// TIA Portal V17 export
// export: Created 2024-09-02T12:49:56.4347094Z, ExportSetting WithDefaults, DisplayName Totally Integrated Automation Portal, DisplayVersion V17, DisplayName TIA Portal Openness, DisplayVersion V17, DisplayName TIA Portal Version Control Interface, DisplayVersion V17, DisplayName STEP 7 Professional, DisplayVersion V17, DisplayName STEP 7 Safety, DisplayVersion V17, DisplayName WinCC Professional, DisplayVersion V17
FUNCTION "SysFC_Type_Change" : Void   // FC260, LAD
TITLE = Type change / Typwechsel
{ S7_Optimized_Access := 'TRUE' }
AUTHOR : OlegFuehrus
FAMILY : Typwechsel
NAME : Typwechsel
VERSION : 0.1
// stored: AutoNumber true, IsIECCheckEnabled false, SetENOAutomatically false, UDAEnableTagReadback false
   VAR_INPUT
      i_Start : Bool;   // Start Auswertung / Start evaluation
      i_Quit : Bool;   // Tywechsel Quitt / Tywechsel Quitt
      i_Reset : Bool;   // Speicher loeschen / Clear memory
      i_Data : Variant;   // Daten (max 64 Byte) / Data (max 64 Byte)
   END_VAR
   VAR_OUTPUT
      "o_Type Change" : Bool;   // Typwechsel / Type change
      "o_no Type Change" : Bool;   // kein Typwechsel / no type change
      "o_Data Fault" : Bool;   // Fehler Parameter / Error Parameter
   END_VAR
   VAR_IN_OUT
      io_IF_TypeChange : "TypeTypeChange";   // Interface Typwechsel / Interface type change
   END_VAR
   VAR_TEMP
      t_VKE0 : Bool;
      t_VKE1 : Bool;
      t_RetVal : Int;
      t_TempDInt : DInt;
      t_DataFault : Bool;
   END_VAR
   VAR_TEMP   // added for the SCL form of the ladder/FBD networks
      _w1 : Bool;
   END_VAR
BEGIN

REGION Network 1: INIT
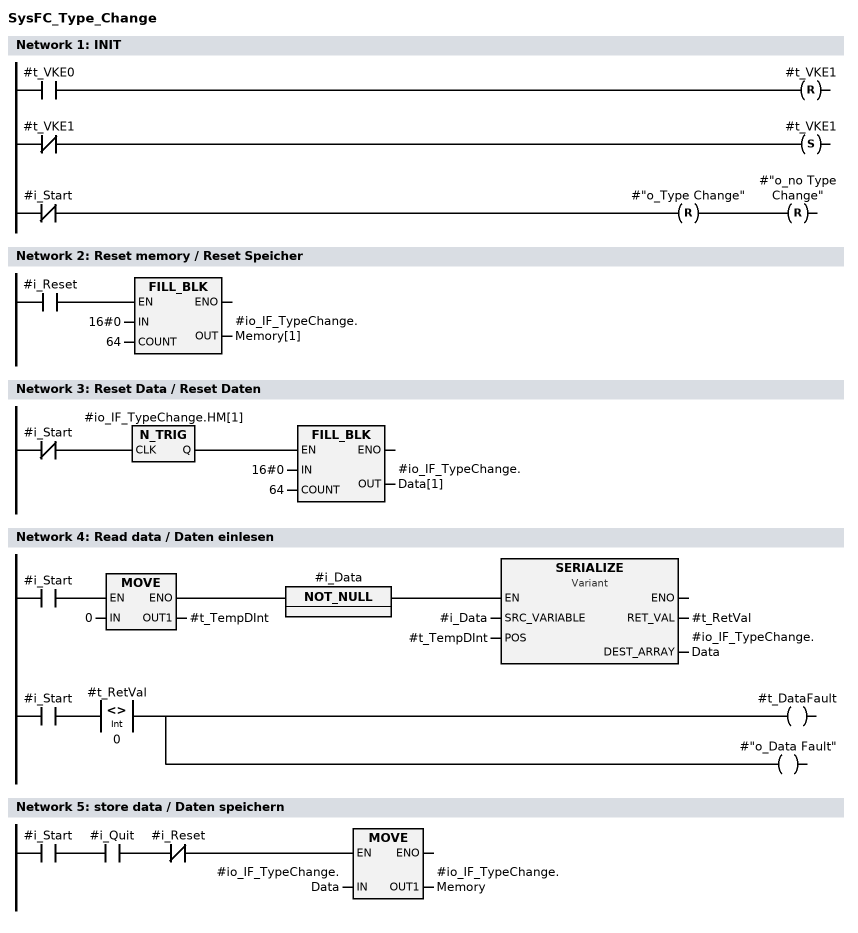
   RUNG wire#powerrail
      Contact( #t_VKE0 )
      R_Coil( #t_VKE1 )
   END_RUNG
   RUNG wire#powerrail
      I_Contact( #t_VKE1 )
      S_Coil( #t_VKE1 )
   END_RUNG
   RUNG wire#powerrail
      I_Contact( #i_Start )
      R_Coil( #"o_Type Change" )
      R_Coil( #"o_no Type Change" )
   END_RUNG
   // the same network as SCL:
   IF #t_VKE0 THEN #t_VKE1 := FALSE; END_IF;
   IF NOT #t_VKE1 THEN #t_VKE1 := TRUE; END_IF;
   IF NOT #i_Start THEN
       #"o_Type Change" := FALSE;
       #"o_no Type Change" := FALSE;
   END_IF;
END_REGION

REGION Network 2: Reset memory / Reset Speicher
   RUNG wire#powerrail
      Contact( #i_Reset )
      FillBlockI(in := 16#0, count := 64, out => #io_IF_TypeChange.Memory[1])
   END_RUNG
   // the same network as SCL:
   IF #i_Reset THEN FILL_BLK(IN := 16#0, COUNT := 64, OUT => #io_IF_TypeChange.Memory[1]); END_IF;
END_REGION

REGION Network 3: Reset Data / Reset Daten
   RUNG wire#powerrail
      I_Contact( #i_Start )
      N_Trig( #io_IF_TypeChange.HM[1] )
      FillBlockI(in := 16#0, count := 64, out => #io_IF_TypeChange.Data[1])
   END_RUNG
   // the same network as SCL:
   #_w1 := NOT (NOT #i_Start) AND #io_IF_TypeChange.HM[1];   // falling edge
   #io_IF_TypeChange.HM[1] := NOT #i_Start;
   IF #_w1 THEN FILL_BLK(IN := 16#0, COUNT := 64, OUT => #io_IF_TypeChange.Data[1]); END_IF;
END_REGION

REGION Network 4: Read data / Daten einlesen
   // no SCL statement known for NOT_NULL: written as a call
   IF #i_Start THEN #t_TempDInt := 0; END_IF;
   IF #i_Start AND NOT_NULL(#i_Data) THEN
       #t_RetVal := Serialize(SRC_VARIABLE := #i_Data, POS := #t_TempDInt, DEST_ARRAY => #io_IF_TypeChange.Data);
   END_IF;
   #t_DataFault := #i_Start AND (#t_RetVal <> 0);
   #"o_Data Fault" := #t_DataFault;
END_REGION

REGION Network 5: store data / Daten speichern
   RUNG wire#powerrail
      Contact( #i_Start )
      Contact( #i_Quit )
      I_Contact( #i_Reset )
      Move(in := #io_IF_TypeChange.Data, out1 => #io_IF_TypeChange.Memory)
   END_RUNG
   // the same network as SCL:
   IF #i_Start AND #i_Quit AND NOT #i_Reset THEN #io_IF_TypeChange.Memory := #io_IF_TypeChange.Data; END_IF;
END_REGION

REGION Network 6 (SCL): Type change / Typwechsel
   IF #i_Start AND NOT #t_DataFault THEN

       IF #io_IF_TypeChange.Data = #io_IF_TypeChange.Memory THEN
           #"o_Type Change" := false;
           #"o_no Type Change" := true;
       ELSE
           #"o_Type Change" := TRUE;
           #"o_no Type Change" := false;
       END_IF;

   END_IF;
END_REGION
END_FUNCTION
